{attribute 'qualified_only'}
{attribute 'strict'}
TYPE E_TIME_SIGNAL_STATUS :
(
	CONNECTED := 0,
	NOT_CONNECTED
);
END_TYPE

(* stored: Version 1.1.0.1, ProductVersion 3.1.4022.12
   DUT E_TIME_SIGNAL_STATUS: Id {7de211d5-5edf-42c9-a1f3-4372dfd33b60} *)
